{attribute 'linkalways'} 
{attribute 'no_explicit_call' := 'This FB is a CLASS and must be accessed using methods or properties'}
{attribute 'enable_dynamic_creation'}
FUNCTION_BLOCK Node_F_VN_InsertIntoContainer_UDINT EXTENDS VisionNode
VAR
    nElement : _UDINT(0);
    ipContainer : _ITcVnContainer;
    nIndex : _ULINT(0);
    hrPrev : _HRESULT(S_OK);
    hresult : _HRESULT(S_OK);
END_VAR

METHOD PUBLIC  Clone : I_Node
VAR
	pNode : POINTER TO Node_F_VN_InsertIntoContainer_UDINT;
END_VAR
pNode := __NEW(Node_F_VN_InsertIntoContainer_UDINT);
Clone := pNode^;
END_METHOD

METHOD FB_init : BOOL
VAR_INPUT
	bInitRetains : BOOL; // if TRUE, the retain variables are initialized (warm start / cold start)
	bInCopyCode : BOOL;  // if TRUE, the instance afterwards gets moved into the copy code (online change)
END_VAR
AddParameter('nElement', nElement);
AddInput('ipContainer', ipContainer);
AddParameter('nIndex', nIndex);
AddInput('hrPrev', hrPrev);
AddOutput('ipContainer', ipContainer);
AddOutput('hresult',hresult);
END_METHOD

METHOD PROTECTED OnExecute
hresult.Value := F_VN_InsertIntoContainer_UDINT(
    nElement := nElement.Value,
    ipContainer := ipContainer.Value,
    nIndex := nIndex.Value,
    hrPrev:= hrPrev.Value);
END_METHOD

METHOD PUBLIC PreExecutionCheck
VAR_INPUT
	Check : I_PreExecutionChecks;
END_VAR
Check.IsTrue(ipContainer.IsValid, 'ipContainer must be a valid container');
Check.IsTrue(ipContainer.IsType(TC_GLOBAL_CONST_LIST.ContainerType_Vector_UDINT), 'ipContainer contains incorrect type');
END_METHOD

END_FUNCTION_BLOCK

(* stored: Version 1.1.0.1, ProductVersion 3.1.4026.13
   POU Node_F_VN_InsertIntoContainer_UDINT: Id {e4308814-9bc5-410b-8556-53c4d3db3a08}, SpecialFunc None
   Folder Constructor: Id {5dbf66df-6851-4944-8548-8e26362a4633}
   Method Clone: Id {3bc6a6f5-7e8c-49a9-a707-3bdf60142e21}
   Method FB_init: Id {56b5300c-cb0e-4877-8208-7f6d3bdd6c7e}
   Method OnExecute: Id {ee757632-770d-4da4-9998-834bfa5a4dd1}
   Method PreExecutionCheck: Id {53ecf133-4786-44e2-b4d4-0d1fb64e62a2} *)
